INTERFACE I_Station EXTENDS __SYSTEM.IQueryInterface

METHOD isComplete : BOOL
VAR_INPUT
END_VAR
END_METHOD

METHOD MyMover : HRESULT
VAR_INPUT
	mover : I_XtsMover;
END_VAR
END_METHOD

PROPERTY Position : MC_LREAL
GET
END_GET
END_PROPERTY

END_INTERFACE

(* stored: Version 1.1.0.1
   Itf I_Station: Id {d8773b48-8571-4ecd-8cbd-ba8942597bd4}
   Method isComplete: Id {60ede7f6-c745-40a4-bf92-f3a03a7a1452}
   Method MyMover: Id {e0d36098-8d65-476a-990c-e6fc9c4a3a40}
   Property Position: Id {382268c5-e001-4500-92a7-4729d1276a58}
   Get Get: Id {419af852-7c98-4df9-a521-739afc5b0cdd} *)
